RoboDK station: trajectories_robolink.rdk

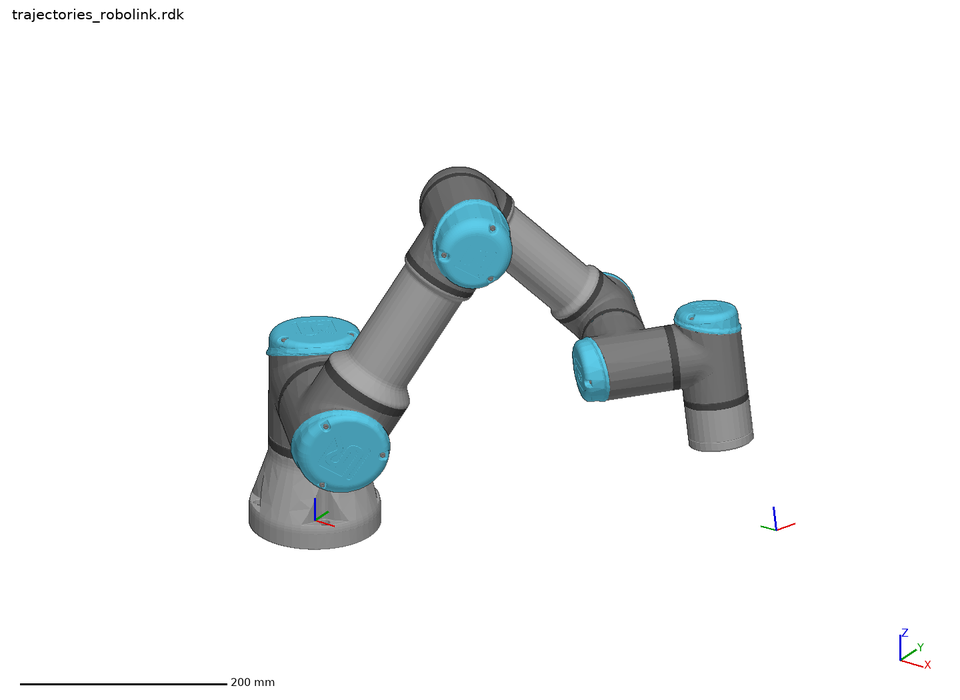
[picture v0: the station drawn from its stored meshes, robots at their saved joint values, targets as dots, program paths as lines]
Station trajectories_robolink (saved by RoboDK 5.6.2). Poses are relative to the parent item; angles as X-Y-Z fixed-axis rotations.
  - frame UR3e Base at (0, 0, 0) mm
    - robot UR3e: 6 axes, payload 3 kg, reach 500 mm, repeatability 0.03 mm, weight 11 kg
        modified DH rows (alpha deg, a mm, theta deg, d mm): 0, 0, 0, 151.9; 90, 0, 180, 0; 0, 243.55, 0, 0; 0, 213.2, 0, 131.05; -90, 0, 0, 85.35; 90, 0, 180, 92.1
        joint limits [-360, -360, -360, -360, -360, -360] to [360, 360, 360, 360, 360, 360]; home [0, -90, -90, 0, 90, 0]; saved at [44.423, -122.178, -102.554, -40.158, 80.889, -121.247]
      - tool TCP_Marker, TCP at (16.91, -17.48, 47.5) mm, rotated rx 180 ry 0 rz 0 deg
    - frame WorkObject at (417, 183, 33) mm, rotated rx -10.43 ry 0.32 rz 75.23 deg
